PROGRAM P_SAFETY
VAR
	Door1_Box	: BOOL;
	Door2_Fence : BOOL;
	Door3_Workbench : BOOL;
	
END_VAR


A_Doors();	// Checking if doors are open
A_Checks(); // Acting on sensor inputs

	//Virtual switches waiting for physical ones
	SAFETY.E_STOP_OK 		:= TRUE;
	GENERAL.Motor_OK		:= TRUE;
	
//============
// If VFD is ready and Security is satisfactory, global "Good To Go"-signal is given
IF GENERAL.Motor_OK AND SAFETY.Safety_OK THEN
	GENERAL.ReadyForAction := TRUE;
END_IF

ACTION A_Checks:
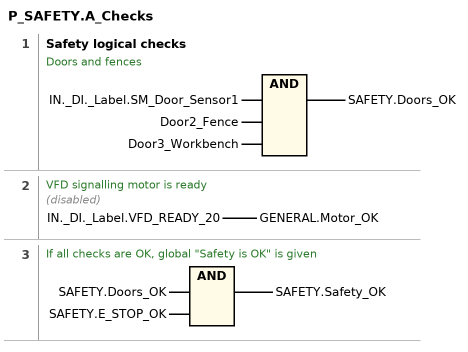
// NETWORK 1: Safety logical checks
// Doors and fences
SAFETY.Doors_OK := IN._DI._Label.SM_Door_Sensor1 AND Door2_Fence AND Door3_Workbench;

// NETWORK 2 (disabled)
// VFD signalling motor is ready
// GENERAL.Motor_OK := IN._DI._Label.VFD_READY_20;

// NETWORK 3
// If all checks are OK, global "Safety is OK" is given
SAFETY.Safety_OK := SAFETY.Doors_OK AND SAFETY.E_STOP_OK;
END_ACTION

ACTION A_Doors:
//"Door sensor" is active Output running to magnet sensor in door
OUT._DO._Label.DoorSensor_Activator := TRUE;

//========================

Door1_Box 		:= IN._DI._Label.SM_Door_Sensor1;	// Previously activated door sensor output is listened here
Door2_Fence 	:= TRUE;							// Not implemented physically	
Door3_Workbench := TRUE;							// Not implemented physically

IF (Door1_Box AND Door2_Fence AND Door3_Workbench) = TRUE THEN	// Checking through all doors and fences
	SAFETY.Doors_OK := TRUE;
	ELSE
		SAFETY.Doors_OK := FALSE;
END_IF
END_ACTION

END_PROGRAM

(* stored: Version 1.1.0.1, ProductVersion 3.1.4024.10
   POU P_SAFETY: Id {4a2af581-3054-4755-8b59-c878439b7ede}, SpecialFunc None
   Action A_Checks: Id {31e58434-104c-4f87-a55e-e4db7b3ddc8a}
   Action A_Doors: Id {3c93ff02-0eab-4dfe-bdea-6020103f9083} *)
